FUNCTION_BLOCK InputSender (* Extracted Composite Function Block Type *)
  (* Version 11/3/2016, Dmitry *)
  PACKAGE Main;
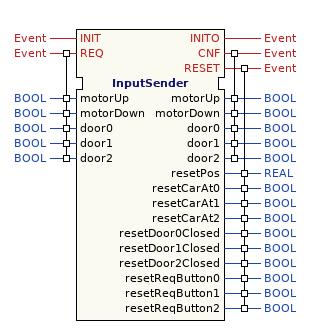
  EVENT_INPUT
    INIT; (* Initialization Request *)
    REQ WITH motorUp, motorDown, door0, door1, door2; (* Normal Execution Request *)
  END_EVENT
  EVENT_OUTPUT
    INITO; (* Initialization Confirm *)
    CNF WITH motorUp, motorDown, door0, door1, door2; (* Execution Confirmation *)
    RESET WITH resetPos, resetCarAt0, resetCarAt1, resetCarAt2, resetDoor0Closed, resetDoor1Closed, resetDoor2Closed, resetReqButton0, resetReqButton1, resetReqButton2;
  END_EVENT
  VAR_INPUT
    motorUp : BOOL;
    motorDown : BOOL;
    door0 : BOOL;
    door1 : BOOL;
    door2 : BOOL;
  END_VAR
  VAR_OUTPUT
    motorUp : BOOL;
    motorDown : BOOL;
    door0 : BOOL;
    door1 : BOOL;
    door2 : BOOL;
    resetPos : REAL;
    resetCarAt0 : BOOL;
    resetCarAt1 : BOOL;
    resetCarAt2 : BOOL;
    resetDoor0Closed : BOOL;
    resetDoor1Closed : BOOL;
    resetDoor2Closed : BOOL;
    resetReqButton0 : BOOL;
    resetReqButton1 : BOOL;
    resetReqButton2 : BOOL;
  END_VAR
  FBS
    FB2 : TCPIO(PORT := ;127.0.0.1:64999);
    FB4 : InputCompressor(delimiter := ;, QI := TRUE);
    FB5 : InputDecompressor(delimiter := ;);
  END_FBS
  EVENT_CONNECTIONS
    FB4.INITO TO FB2.INIT;
    INIT TO FB4.INIT;
    REQ TO FB4.REQ;
    FB4.CNF TO FB2.REQ;
    FB2.CNF TO FB2.ACK;
    FB2.IND TO FB5.REQ;
    FB2.INITO TO FB5.INIT;
    FB5.INITO TO INITO;
    FB5.CNF TO CNF;
    FB5.RESET TO RESET;
  END_CONNECTIONS
  DATA_CONNECTIONS
    FB4.QO TO FB2.QI;
    FB5.motorUp TO motorUp;
    FB5.motorDown TO motorDown;
    FB5.door0 TO door0;
    FB5.door1 TO door1;
    FB5.door2 TO door2;
    motorUp TO FB4.motorUp;
    motorDown TO FB4.motorDown;
    door0 TO FB4.door0;
    door1 TO FB4.door1;
    door2 TO FB4.door2;
    FB4.RESULT TO FB2.DATAOUT;
    FB2.DATAIN TO FB5.input;
    FB2.QO TO FB5.QI;
    FB5.resetPos TO resetPos;
    FB5.resetCarAt0 TO resetCarAt0;
    FB5.resetCarAt1 TO resetCarAt1;
    FB5.resetCarAt2 TO resetCarAt2;
    FB5.resetDoor1Closed TO resetDoor1Closed;
    FB5.resetDoor2Closed TO resetDoor2Closed;
    FB5.resetReqButton0 TO resetReqButton0;
    FB5.resetDoor0Closed TO resetDoor0Closed;
    FB5.resetReqButton1 TO resetReqButton1;
    FB5.resetReqButton2 TO resetReqButton2;
  END_CONNECTIONS
END_FUNCTION_BLOCK
